// Mitsubishi GX Works2 project: WashingMachine   PLC: FX2N/FX2NC

PROGRAM MAIN
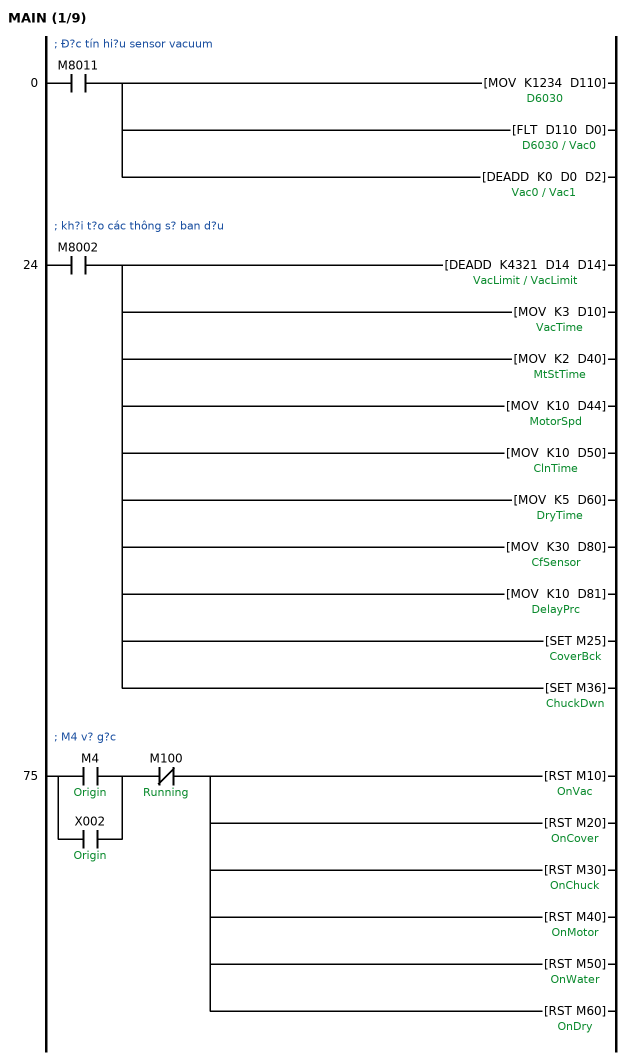
; Ð?c tín hi?u sensor vacuum
; 
0     LD      M8011
      MOV     K1234 D110  ; D6030
      FLT     D110 D0  ; Vac0
      DEADD   K0 D0 D2  ; Vac1
; kh?i t?o các thông s? ban d?u
24    LD      M8002
      DEADD   K4321 D14 D14  ; VacLimit
      MOV     K3 D10  ; VacTime
      MOV     K2 D40  ; MtStTime
      MOV     K10 D44  ; MotorSpd
      MOV     K10 D50  ; ClnTime
      MOV     K5 D60  ; DryTime
      MOV     K30 D80  ; CfSensor
      MOV     K10 D81  ; DelayPrc
      SET     M25  ; CoverBck
      SET     M36  ; ChuckDwn
; M4 v? g?c
75    LD      M4  ; Origin
      OR      X002  ; Origin
      ANI     M100  ; Running
      RST     M10  ; OnVac
      RST     M20  ; OnCover
      RST     M30  ; OnChuck
      RST     M40  ; OnMotor
      RST     M50  ; OnWater
      RST     M60  ; OnDry
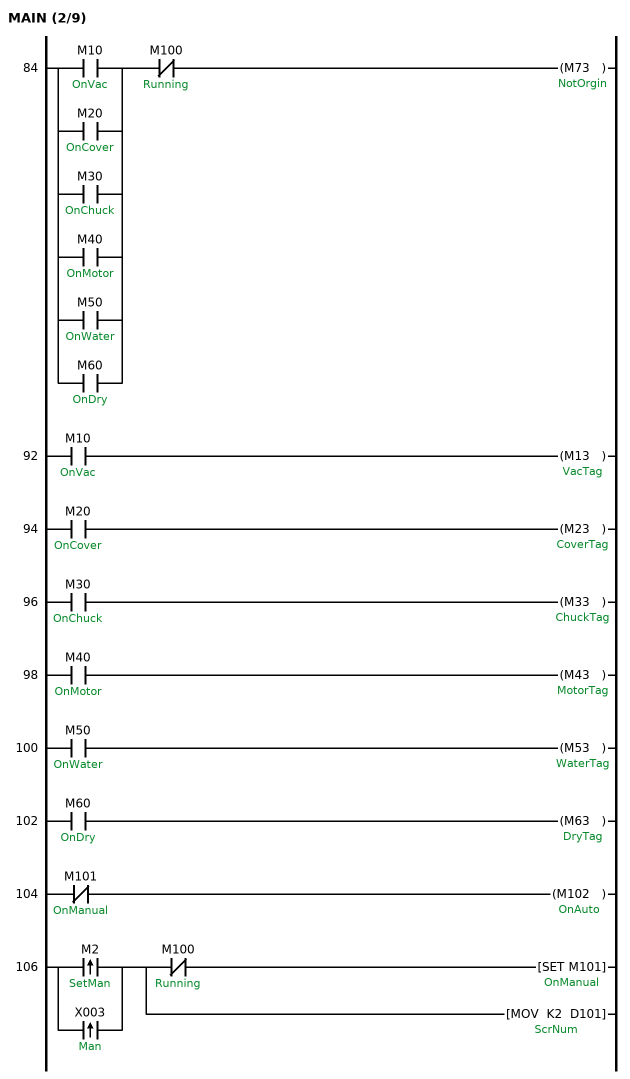
84    LD      M10  ; OnVac
      OR      M20  ; OnCover
      OR      M30  ; OnChuck
      OR      M40  ; OnMotor
      OR      M50  ; OnWater
      OR      M60  ; OnDry
      ANI     M100  ; Running
      OUT     M73  ; NotOrgin
92    LD      M10  ; OnVac
      OUT     M13  ; VacTag
94    LD      M20  ; OnCover
      OUT     M23  ; CoverTag
96    LD      M30  ; OnChuck
      OUT     M33  ; ChuckTag
98    LD      M40  ; OnMotor
      OUT     M43  ; MotorTag
100   LD      M50  ; OnWater
      OUT     M53  ; WaterTag
102   LD      M60  ; OnDry
      OUT     M63  ; DryTag
104   LDI     M101  ; OnManual
      OUT     M102  ; OnAuto
106   LDP     M2  ; SetMan
      ORP     X003  ; Man
      MPS
      ANI     M100  ; Running
      SET     M101  ; OnManual
      MPP
      MOV     K2 D101  ; ScrNum
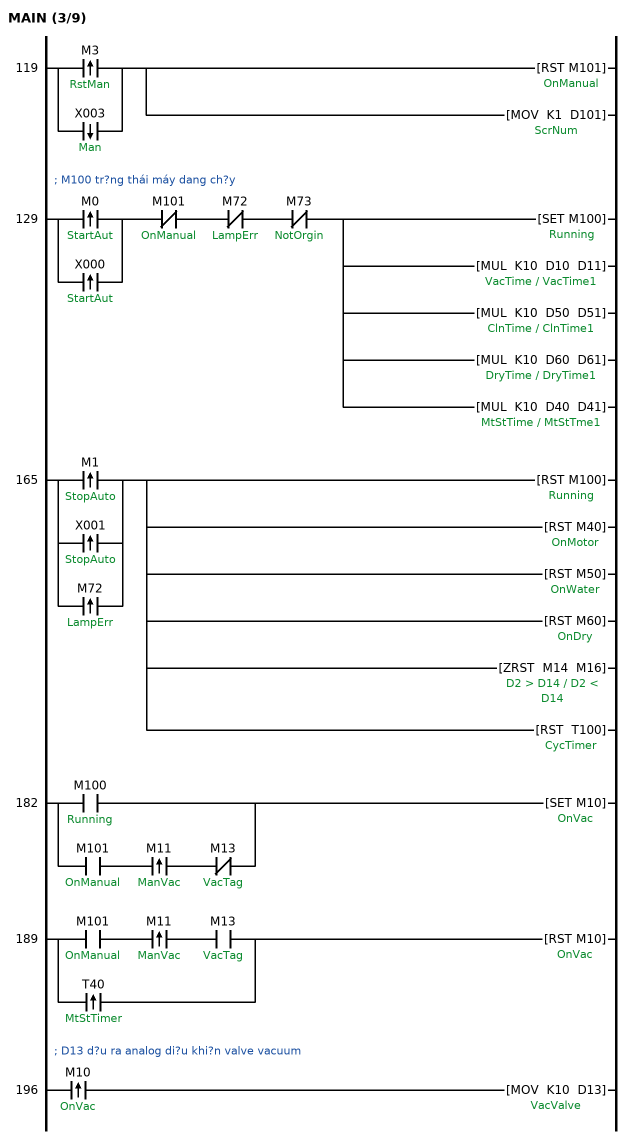
119   LDP     M3  ; RstMan
      ORF     X003  ; Man
      RST     M101  ; OnManual
      MOV     K1 D101
; M100 tr?ng thái máy dang ch?y
129   LDP     M0  ; StartAut
      ORP     X000  ; StartAut
      ANI     M101  ; OnManual
      ANI     M72  ; LampErr
      ANI     M73  ; NotOrgin
      SET     M100  ; Running
      MUL     K10 D10 D11  ; VacTime1
      MUL     K10 D50 D51  ; ClnTime1
      MUL     K10 D60 D61  ; DryTime1
      MUL     K10 D40 D41  ; MtStTme1
165   LDP     M1  ; StopAuto
      ORP     X001  ; StopAuto
      ORP     M72  ; LampErr
      RST     M100  ; Running
      RST     M40  ; OnMotor
      RST     M50  ; OnWater
      RST     M60  ; OnDry
      ZRST    M14 M16  ; D2 > D14 / D2 < D14
      RST     T100  ; CycTimer
182   LD      M100  ; Running
      LD      M101  ; OnManual
      ANDP    M11  ; ManVac
      ANI     M13  ; VacTag
      ORB
      SET     M10  ; OnVac
189   LD      M101  ; OnManual
      ANDP    M11  ; ManVac
      AND     M13  ; VacTag
      ORP     T40  ; MtStTimer
      RST     M10  ; OnVac
; D13 d?u ra analog di?u khi?n valve vacuum
196   LDP     M10  ; OnVac
      MOV     K10 D13  ; VacValve
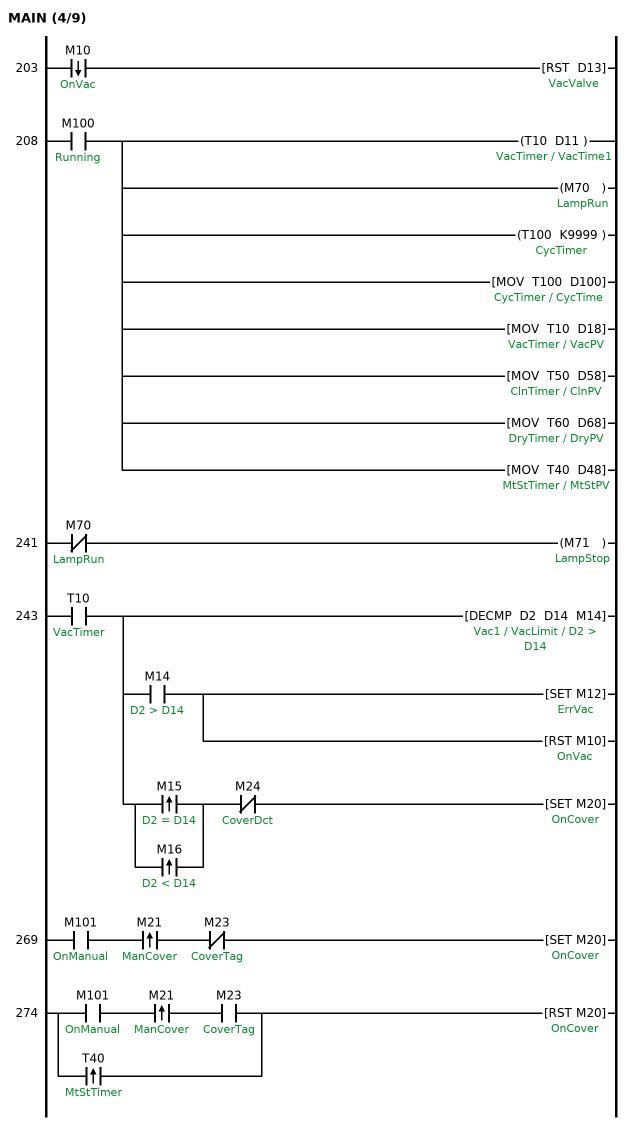
203   LDF     M10  ; OnVac
      RST     D13  ; VacValve
208   LD      M100  ; Running
      OUT     T10 D11  ; VacTimer / VacTime1
      OUT     M70  ; LampRun
      OUT     T100 K9999  ; CycTimer
      MOV     T100 D100  ; CycTime
      MOV     T10 D18  ; VacPV
      MOV     T50 D58  ; ClnTimer / ClnPV
      MOV     T60 D68  ; DryTimer / DryPV
      MOV     T40 D48  ; MtStPV
241   LDI     M70  ; LampRun
      OUT     M71  ; LampStop
243   LD      T10  ; VacTimer
      DECMP   D2 D14 M14
      MPS
      AND     M14  ; D2 > D14
      SET     M12  ; ErrVac
      RST     M10  ; OnVac
      MPP
      LDP     M15  ; D2 = D14
      ORP     M16  ; D2 < D14
      ANB
      ANI     M24  ; CoverDct
      SET     M20  ; OnCover
269   LD      M101  ; OnManual
      ANDP    M21  ; ManCover
      ANI     M23  ; CoverTag
      SET     M20  ; OnCover
274   LD      M101  ; OnManual
      ANDP    M21  ; ManCover
      AND     M23  ; CoverTag
      ORP     T40  ; MtStTimer
      RST     M20  ; OnCover
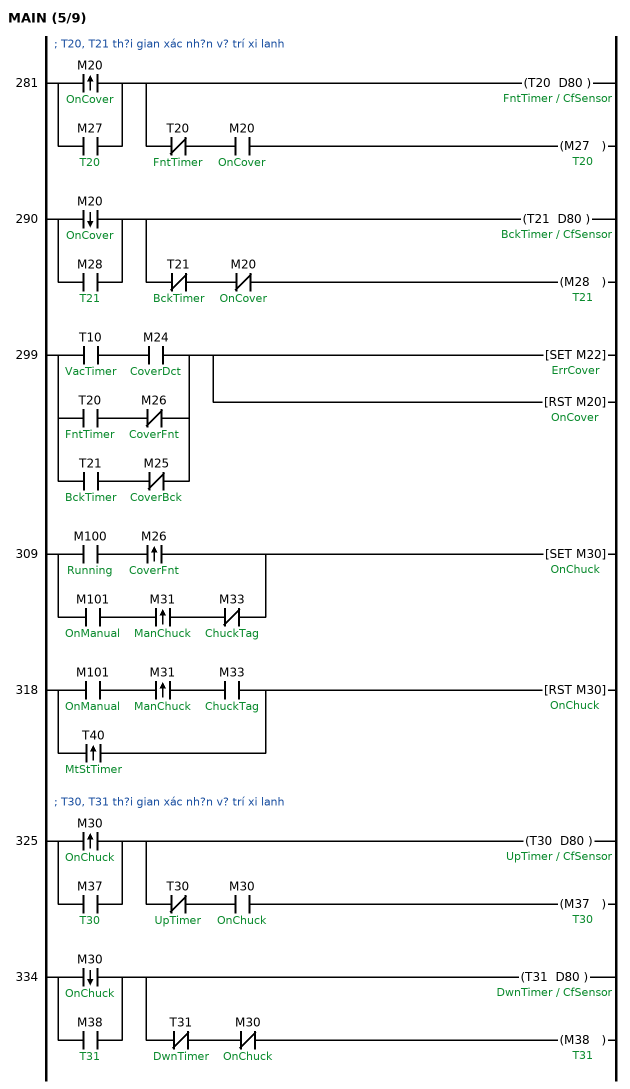
; T20, T21 th?i gian xác nh?n v? trí xi lanh
281   LDP     M20  ; OnCover
      OR      M27  ; T20
      OUT     T20 D80  ; FntTimer / CfSensor
      ANI     T20  ; FntTimer
      AND     M20  ; OnCover
      OUT     M27  ; T20
290   LDF     M20  ; OnCover
      OR      M28  ; T21
      OUT     T21 D80  ; BckTimer / CfSensor
      ANI     T21  ; BckTimer
      ANI     M20  ; OnCover
      OUT     M28  ; T21
299   LD      T10  ; VacTimer
      AND     M24  ; CoverDct
      LD      T20  ; FntTimer
      ANI     M26  ; CoverFnt
      ORB
      LD      T21  ; BckTimer
      ANI     M25  ; CoverBck
      ORB
      SET     M22  ; ErrCover
      RST     M20  ; OnCover
309   LD      M100  ; Running
      ANDP    M26  ; CoverFnt
      LD      M101  ; OnManual
      ANDP    M31  ; ManChuck
      ANI     M33  ; ChuckTag
      ORB
      SET     M30  ; OnChuck
318   LD      M101  ; OnManual
      ANDP    M31  ; ManChuck
      AND     M33  ; ChuckTag
      ORP     T40  ; MtStTimer
      RST     M30  ; OnChuck
; T30, T31 th?i gian xác nh?n v? trí xi lanh
325   LDP     M30  ; OnChuck
      OR      M37  ; T30
      OUT     T30 D80  ; UpTimer / CfSensor
      ANI     T30  ; UpTimer
      AND     M30  ; OnChuck
      OUT     M37  ; T30
334   LDF     M30  ; OnChuck
      OR      M38  ; T31
      OUT     T31 D80  ; DwnTimer / CfSensor
      ANI     T31  ; DwnTimer
      ANI     M30  ; OnChuck
      OUT     M38  ; T31
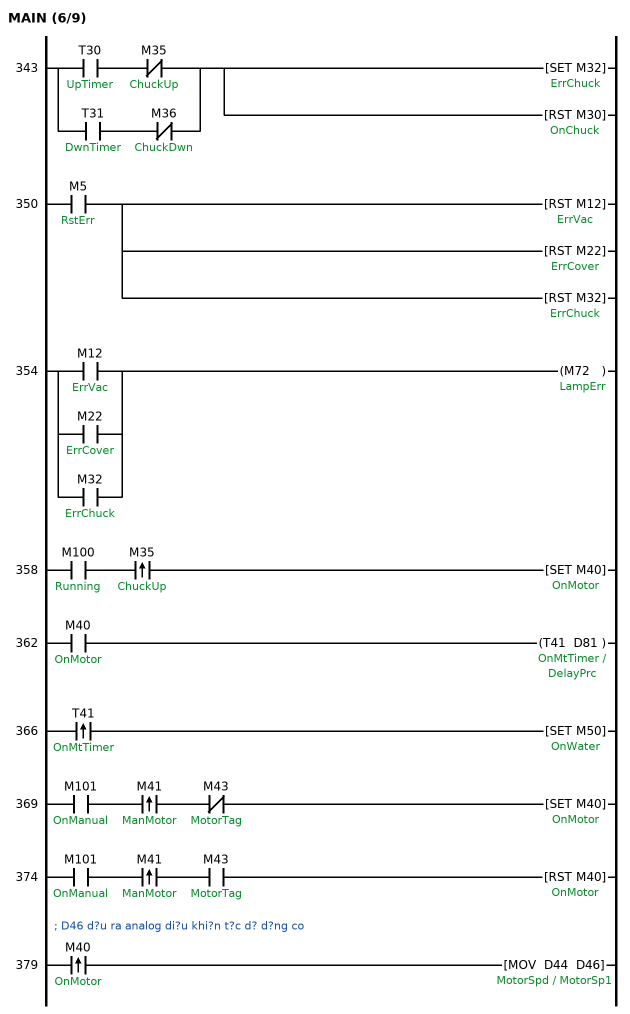
343   LD      T30  ; UpTimer
      ANI     M35  ; ChuckUp
      LD      T31  ; DwnTimer
      ANI     M36  ; ChuckDwn
      ORB
      SET     M32  ; ErrChuck
      RST     M30  ; OnChuck
350   LD      M5  ; RstErr
      RST     M12  ; ErrVac
      RST     M22  ; ErrCover
      RST     M32  ; ErrChuck
354   LD      M12  ; ErrVac
      OR      M22  ; ErrCover
      OR      M32  ; ErrChuck
      OUT     M72  ; LampErr
358   LD      M100  ; Running
      ANDP    M35  ; ChuckUp
      SET     M40  ; OnMotor
362   LD      M40  ; OnMotor
      OUT     T41 D81  ; OnMtTimer / DelayPrc
366   LDP     T41  ; OnMtTimer
      SET     M50  ; OnWater
369   LD      M101  ; OnManual
      ANDP    M41  ; ManMotor
      ANI     M43  ; MotorTag
      SET     M40  ; OnMotor
374   LD      M101  ; OnManual
      ANDP    M41  ; ManMotor
      AND     M43  ; MotorTag
      RST     M40  ; OnMotor
; D46 d?u ra analog di?u khi?n t?c d? d?ng co
379   LDP     M40  ; OnMotor
      MOV     D44 D46  ; MotorSp1
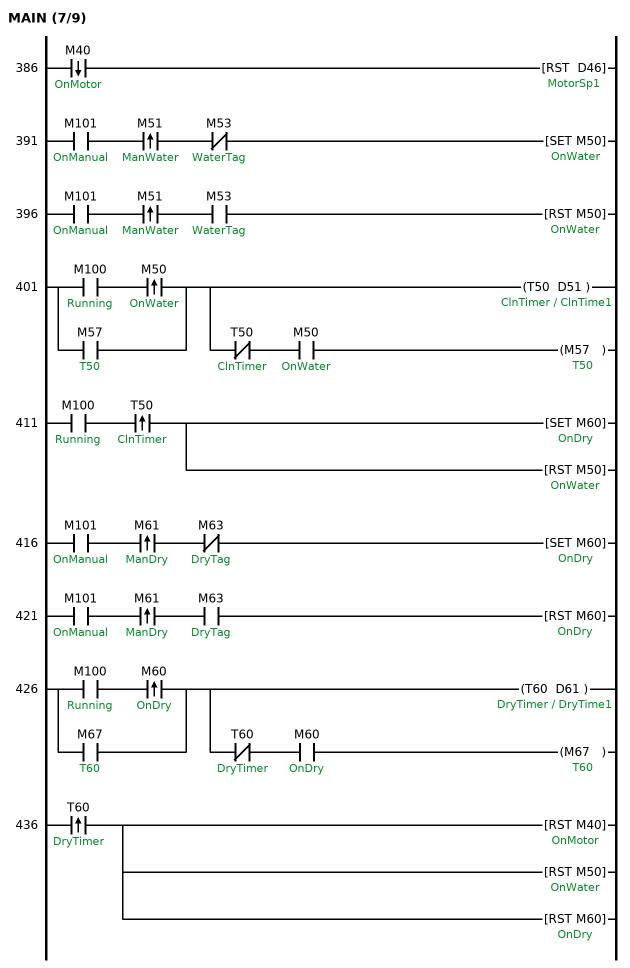
386   LDF     M40  ; OnMotor
      RST     D46  ; MotorSp1
391   LD      M101  ; OnManual
      ANDP    M51  ; ManWater
      ANI     M53  ; WaterTag
      SET     M50  ; OnWater
396   LD      M101  ; OnManual
      ANDP    M51  ; ManWater
      AND     M53  ; WaterTag
      RST     M50  ; OnWater
401   LD      M100  ; Running
      ANDP    M50  ; OnWater
      OR      M57  ; T50
      OUT     T50 D51  ; ClnTimer / ClnTime1
      ANI     T50  ; ClnTimer
      AND     M50  ; OnWater
      OUT     M57  ; T50
411   LD      M100  ; Running
      ANDP    T50  ; ClnTimer
      SET     M60  ; OnDry
      RST     M50  ; OnWater
416   LD      M101  ; OnManual
      ANDP    M61  ; ManDry
      ANI     M63  ; DryTag
      SET     M60  ; OnDry
421   LD      M101  ; OnManual
      ANDP    M61  ; ManDry
      AND     M63  ; DryTag
      RST     M60  ; OnDry
426   LD      M100  ; Running
      ANDP    M60  ; OnDry
      OR      M67  ; T60
      OUT     T60 D61  ; DryTimer / DryTime1
      ANI     T60  ; DryTimer
      AND     M60  ; OnDry
      OUT     M67  ; T60
436   LDP     T60  ; DryTimer
      RST     M40  ; OnMotor
      RST     M50  ; OnWater
      RST     M60  ; OnDry
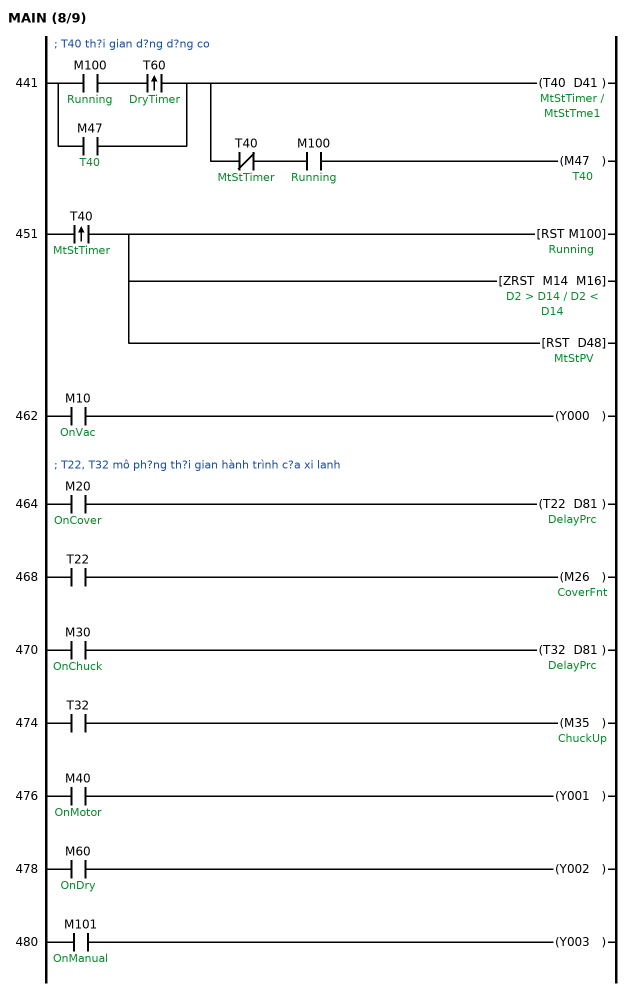
; T40 th?i gian d?ng d?ng co
441   LD      M100  ; Running
      ANDP    T60  ; DryTimer
      OR      M47  ; T40
      OUT     T40 D41  ; MtStTimer / MtStTme1
      ANI     T40  ; MtStTimer
      AND     M100  ; Running
      OUT     M47  ; T40
451   LDP     T40  ; MtStTimer
      RST     M100  ; Running
      ZRST    M14 M16
      RST     D48  ; MtStPV
462   LD      M10  ; OnVac
      OUT     Y000
; T22, T32 mô ph?ng th?i gian hành trình c?a xi lanh
464   LD      M20  ; OnCover
      OUT     T22 D81  ; DelayPrc
468   LD      T22
      OUT     M26  ; CoverFnt
470   LD      M30  ; OnChuck
      OUT     T32 D81  ; DelayPrc
474   LD      T32
      OUT     M35  ; ChuckUp
476   LD      M40  ; OnMotor
      OUT     Y001
478   LD      M60  ; OnDry
      OUT     Y002
480   LD      M101  ; OnManual
      OUT     Y003
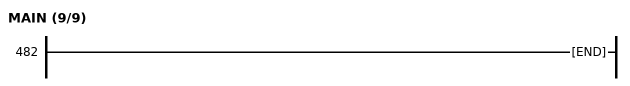
482   END
END_PROGRAM
